// Mitsubishi GX Works2 project: flipflop   PLC: Q02/Q02H

PROGRAM MAIN
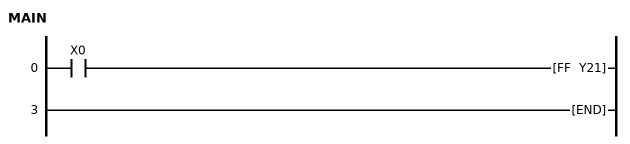
0     LD      X0
      FF      Y21
3     END
END_PROGRAM
